{attribute 'qualified_only'}
VAR_GLOBAL
        
    {attribute 'pytmc' := '
     pv: MR1K4:SOMS:MMS:YUP:STATE;
     io: io;
    '}
    fbMR1K4_Coating_States: FB_Coating_States_noPMPS; 
    
    MR1K4_SiC : DUT_PositionState := (
        bUseRawCounts := TRUE,
        bMoveOk := TRUE,
        bValid := TRUE,
        sName := 'SiC',  
        nEncoderCount := 22000532,
        fDelta := 1000,
        fVelocity := 150);
        
    MR1K4_B4C : DUT_PositionState := (
        bUseRawCounts := TRUE,
        bMoveOk := TRUE,
        bValid := TRUE,
        sName := 'B4C',  
        nEncoderCount := 5000141,
        fDelta := 1000,
        fVelocity := 150);
            
    {attribute 'pytmc' := '
     pv: MR2K4:KBO:MMS:Y:STATE;
     io: io;
    '}
    fbMR2K4_Coating_States: FB_Coating_States_noPMPS; 
    
    MR2K4_SiC : DUT_PositionState := (
        bUseRawCounts := TRUE,
        bMoveOk := TRUE,
        bValid := TRUE,
        sName := 'SiC',  
        nEncoderCount := 8701960,
        fDelta := 1,
        fVelocity := 0.150);
        
    MR2K4_B4C : DUT_PositionState := (
        bUseRawCounts := TRUE,
        bMoveOk := TRUE,
        bValid := TRUE,
        sName := 'B4C',  
        nEncoderCount := 6636177,
        fDelta := 1,
        fVelocity := 0.150);
    {attribute 'pytmc' := '
     pv: MR3K4:KBO:MMS:X:STATE;
     io: io;
    '}
    fbMR3K4_Coating_States: FB_Coating_States_noPMPS; 
    
    MR3K4_SiC : DUT_PositionState := (
        bUseRawCounts := TRUE,
        bMoveOk := TRUE,
        bValid := TRUE,
        sName := 'SiC',  
        nEncoderCount := 4719890,
        fDelta := 1,
        fVelocity := 0.150);
        
    MR3K4_B4C : DUT_PositionState := (
        bUseRawCounts := TRUE,
        bMoveOk := TRUE,
        bValid := TRUE,
        sName := 'B4C',  
        nEncoderCount := 8220029,
        fDelta := 1,
        fVelocity := 0.150);
END_VAR

(* stored: Version 1.1.0.1, ProductVersion 3.1.4022.18
   GVL GVL_States: Id {11a005be-0297-4fb5-969c-f097945fdbd4} *)
